PROGRAM Valvulas
VAR

(*=========================		VÁLVULAS		==========================*)	



(*========================================================================*)

END_VAR

(*==============		Válvula Y1 - XXXXXXX XXXXXXX		==============*)

IF (MaquinaModoManual) THEN
	//Controle Manual - Válvula Y1
	IF (IhmBt_Y1_Ligar) THEN
		OutValvulaY1R := FALSE;	//Solenóide de Recuo
		OutValvulaY1A := TRUE; //Solenóide de Avanço
	ELSE
		OutValvulaY1A := FALSE;	//Solenóide de Avanço
		OutValvulaY1R := TRUE; //Solenóide de Recuo	
	END_IF
ELSIF (MaquinaModoAuto) THEN
	//Controle Automático - Válvula Y1
	IF (AvancarValvulaY1) THEN
		OutValvulaY1R := FALSE; //Solenóide de Recuo
		OutValvulaY1A := TRUE;	//Solenóide de Avanço
	ELSE
		OutValvulaY1A := FALSE; //Solenóide de Avanço
		OutValvulaY1R := TRUE;	//Solenóide de Recuo
	END_IF
ELSE
	OutValvulaY1R := FALSE; //Solenóide de Recuo
	OutValvulaY1A := FALSE;	//Solenóide de Avanço
END_IF

(*========================================================================*)

(*==============		Válvula Y2 - XXXXXXX XXXXXXX		==============*)

IF (MaquinaModoManual) THEN
	//Controle Manual - Válvula Y2
	IF (IhmBt_Y2_Ligar) THEN
		OutValvulaY2R := FALSE;	//Solenóide de Recuo
		OutValvulaY2A := TRUE; //Solenóide de Avanço
	ELSE
		OutValvulaY2A := FALSE;	//Solenóide de Avanço
		OutValvulaY2R := TRUE; //Solenóide de Recuo	
	END_IF
ELSIF (MaquinaModoAuto) THEN
	//Controle Automático - Válvula Y2
	IF (AvancarValvulaY2) THEN
		OutValvulaY2R := FALSE; //Solenóide de Recuo
		OutValvulaY2A := TRUE;	//Solenóide de Avanço
	ELSE
		OutValvulaY2A := FALSE; //Solenóide de Avanço
		OutValvulaY2R := TRUE;	//Solenóide de Recuo
	END_IF
ELSE
	OutValvulaY2R := FALSE; //Solenóide de Recuo
	OutValvulaY2A := FALSE;	//Solenóide de Avanço
END_IF

(*========================================================================*)

(*==============		Válvula Y3 - XXXXXXX XXXXXXX		==============*)

IF (MaquinaModoManual) THEN
	//Controle Manual - Válvula Y3
	IF (IhmBt_Y3_Ligar) THEN
		OutValvulaY3R := FALSE;	//Solenóide de Recuo
		OutValvulaY3A := TRUE; //Solenóide de Avanço
	ELSE
		OutValvulaY3A := FALSE;	//Solenóide de Avanço
		OutValvulaY3R := TRUE; //Solenóide de Recuo	
	END_IF
ELSIF (MaquinaModoAuto) THEN
	//Controle Automático - Válvula Y3
	IF (AvancarValvulaY3) THEN
		OutValvulaY3R := FALSE; //Solenóide de Recuo
		OutValvulaY3A := TRUE;	//Solenóide de Avanço
	ELSE
		OutValvulaY3A := FALSE; //Solenóide de Avanço
		OutValvulaY3R := TRUE;	//Solenóide de Recuo
	END_IF
ELSE
	OutValvulaY3R := FALSE; //Solenóide de Recuo
	OutValvulaY3A := FALSE;	//Solenóide de Avanço
END_IF

(*========================================================================*)

(*==============		Válvula Y4 - XXXXXXX XXXXXXX		==============*)

IF (MaquinaModoManual) THEN
	//Controle Manual - Válvula Y4
	IF (IhmBt_Y4_Ligar) THEN
		OutValvulaY4R := FALSE;	//Solenóide de Recuo
		OutValvulaY4A := TRUE; //Solenóide de Avanço
	ELSE
		OutValvulaY4A := FALSE;	//Solenóide de Avanço
		OutValvulaY4R := TRUE; //Solenóide de Recuo	
	END_IF
ELSIF (MaquinaModoAuto) THEN
	//Controle Automático - Válvula Y4
	IF (AvancarValvulaY4) THEN
		OutValvulaY4R := FALSE; //Solenóide de Recuo
		OutValvulaY4A := TRUE;	//Solenóide de Avanço
	ELSE
		OutValvulaY4A := FALSE; //Solenóide de Avanço
		OutValvulaY4R := TRUE;	//Solenóide de Recuo
	END_IF
ELSE
	OutValvulaY4R := FALSE; //Solenóide de Recuo
	OutValvulaY4A := FALSE;	//Solenóide de Avanço
END_IF

(*========================================================================*)

(*==============		Válvula Y5 - XXXXXXX XXXXXXX		==============*)

IF (MaquinaModoManual) THEN
	//Controle Manual - Válvula Y5
	IF (IhmBt_Y5_Ligar) THEN
		OutValvulaY5R := FALSE;	//Solenóide de Recuo
		OutValvulaY5A := TRUE; //Solenóide de Avanço
	ELSE
		OutValvulaY5A := FALSE;	//Solenóide de Avanço
		OutValvulaY5R := TRUE; //Solenóide de Recuo	
	END_IF
ELSIF (MaquinaModoAuto) THEN
	//Controle Automático - Válvula Y5
	IF (AvancarValvulaY5) THEN
		OutValvulaY5R := FALSE; //Solenóide de Recuo
		OutValvulaY5A := TRUE;	//Solenóide de Avanço
	ELSE
		OutValvulaY5A := FALSE; //Solenóide de Avanço
		OutValvulaY5R := TRUE;	//Solenóide de Recuo
	END_IF
ELSE
	OutValvulaY5R := FALSE; //Solenóide de Recuo
	OutValvulaY5A := FALSE;	//Solenóide de Avanço
END_IF

(*========================================================================*)

(*==============		Válvula Y6 - XXXXXXX XXXXXXX		==============*)

IF (MaquinaModoManual) THEN
	//Controle Manual - Válvula Y6
	IF (IhmBt_Y6_Ligar) THEN
		OutValvulaY6 := TRUE;
	ELSE
		OutValvulaY6 := FALSE;
	END_IF
ELSIF (MaquinaModoAuto) THEN
	//Controle Automático - Válvula Y6
	IF (LigarValvulaY6) THEN
		OutValvulaY6 := TRUE;
	ELSE
		OutValvulaY6 := FALSE;
	END_IF
ELSE
	OutValvulaY6 := FALSE;
END_IF

(*========================================================================*)

(*==============		Válvula Y9 - XXXXXXX XXXXXXX		==============*)

IF (MaquinaModoManual) THEN
	//Controle Manual - Válvula Y9
	IF (IhmBt_Y9_Ligar) THEN
		OutValvulaY9 := TRUE;
	ELSE
		OutValvulaY9 := FALSE;
	END_IF
ELSIF (MaquinaModoAuto) THEN
	//Controle Automático - Válvula Y9
	IF (LigarValvulaY9) THEN
		OutValvulaY9 := TRUE;
	ELSE
		OutValvulaY9 := FALSE;
	END_IF
ELSE
	OutValvulaY9 := FALSE;
END_IF

(*========================================================================*)

(*==========		Válvula Proporcional - XXXXXXX XXXXXXX		==========*)

IF (MaquinaModoManual) THEN
	//Controle Manual - Válvula Proporcional
	IF (IhmBt_VP_Teste) THEN
		ValvulaProporcional := (INT_TO_REAL(IhmEscr_ValvulaProporcional)/100)*(32767);
	END_IF
ELSIF (MaquinaModoAuto) THEN
	//Controle Automático - Válvula Proporcional
	ValvulaProporcional := (INT_TO_REAL(50)/100)*(32767);
ELSE
	ValvulaProporcional := 0;
END_IF
	
(*========================================================================*)

(*=============		Válvula Y7 - Válvula de Segurança 1		==============*)

//Controle Automático - Válvula Y7
IF (NOT Alarmes.AlarmeGrave) THEN
	LigarValvulaY7 := TRUE;
ELSE
	LigarValvulaY7 := FALSE;
END_IF

//Válvula Y7 - XXXXX XXXXX
IF (LigarValvulaY7) THEN
	OutValvulaY7 := TRUE;
ELSE
	OutValvulaY7 := FALSE;
END_IF

(*========================================================================*) 

(*=============		Válvula Y8 - Válvula de Segurança 2		==============*)

//Controle Automático - Válvula Y8
IF (NOT Alarmes.AlarmeGrave) THEN
	LigarValvulaY8 := TRUE;
ELSE
	LigarValvulaY8 := FALSE;
END_IF

//Válvula Y8 - XXXXX XXXXX
IF (LigarValvulaY8) THEN
	OutValvulaY8 := TRUE;
ELSE
	OutValvulaY8 := FALSE;
END_IF

(*========================================================================*)

END_PROGRAM

(* stored: Version 1.1.0.1, ProductVersion 3.1.4024.11
   POU Valvulas: Id {54ed8504-3266-4bd1-b116-5b79c5790bc6}, SpecialFunc None *)
